# EPICS autosave request: iocBoot/sioc-esb-xps2/xps.req
file xpsm.req P=ESB:XPS2:m1
file xpsm.req P=ESB:XPS2:m2
file xpsm.req P=ESB:XPS2:m3
file xpsm.req P=ESB:XPS2:m4
file xpsm.req P=ESB:XPS2:m5
file xpsm.req P=ESB:XPS2:m6
file xpsm.req P=ESB:XPS2:m7
file xpsm.req P=ESB:XPS2:m8
